// TIA Portal V15.1 export
// export: Created 2026-01-09T13:45:11.9352339Z, ExportSetting WithDefaults, WithReadOnly, DisplayName Totally Integrated Automation Portal, DisplayVersion V15.1 Update 8, DisplayName TIA Portal Openness, DisplayVersion V15.1 Update 8, DisplayName STEP 7 Professional, DisplayVersion V15.1 Update 8, DisplayName WinCC Advanced, DisplayVersion V15.1 Update 8
FUNCTION_BLOCK "1.ANALOG_INPUT"   // FB1, LAD
{ S7_Optimized_Access := 'TRUE' }
VERSION : 0.1
// stored: AutoNumber false, CodeModifiedDate 2025-09-22T19:33:21.555545Z, CompileDate 2025-09-22T19:33:35.8164831Z, CreationDate 2024-10-12T12:36:08.0193576Z, DownloadWithoutReinit false, HandleErrorsWithinBlock false, InterfaceModifiedDate 2025-09-22T19:30:11.8403437Z, IsConsistent true, IsIECCheckEnabled false, IsKnowHowProtected false, IsRetainMemResEnabled false, IsWriteProtected false, LibraryConformanceStatus The object is library-conformant., MemoryReserve 100, ModifiedDate 2025-09-22T19:33:21.555545Z, ParameterModified 2025-08-30T17:31:01.4104373Z, PLCSimAdvancedSupport false, SetENOAutomatically False, StructureModified 2025-09-22T19:30:11.8403437Z, UDAEnableTagReadback false
   VAR_INPUT
      AI : Int;
      A_MODE : Real;
      ZERO : Real;
      SPAN : Real;
      BT_ZERO : Bool;
      BT_SPAN : Bool;
      B_MANUAL : Real;
      HMI_Manual_Trigger : Bool;
   END_VAR
   VAR_OUTPUT
      W_OUT : Real;
      X_OUT : Real;
   END_VAR
   VAR RETAIN
      T_AI { ExternalAccessible := 'False'; ExternalVisible := 'False'; ExternalWritable := 'False'} : Real;
      T_AN { ExternalAccessible := 'False'; ExternalVisible := 'False'; ExternalWritable := 'False'} : Real;
      T_ZERO { ExternalAccessible := 'False'; ExternalVisible := 'False'; ExternalWritable := 'False'} : Real;
      AN_ZERO { ExternalAccessible := 'False'; ExternalVisible := 'False'; ExternalWritable := 'False'} : Real;
      T_SPAN { ExternalAccessible := 'False'; ExternalVisible := 'False'; ExternalWritable := 'False'} : Real;
      AN_SPAN { ExternalAccessible := 'False'; ExternalVisible := 'False'; ExternalWritable := 'False'} : Real;
   END_VAR
   VAR
      B_MANUAL_SAVED : Real;
      B_HAS_CHANGED : Bool;
   END_VAR
   VAR RETAIN
      IS_MANUAL_MODE : Bool;
   END_VAR
   VAR
      BT_ZERO_Raising : Bool;
      BT_SPAN_Riasing : Bool;
      MANUAL_Raissing : Bool;
      Bit_Reset_Man_Mode : Bool;
   END_VAR
   VAR_TEMP
      AI_MIN : Int;
      AI_MAX : Int;
      AN_MIN : Real;
      AN_MAX : Real;
      GT_INTEGER : DInt;
      TEMP_RESULT_DINT : DInt;
      W_OUT_MANUAL : Real;
      W_OUT_AUTO : Real;
   END_VAR
   VAR_TEMP   // added for the SCL form of the ladder/FBD networks
      _w1 : Bool;
   END_VAR
BEGIN

REGION Network 1: ANALOG MODE
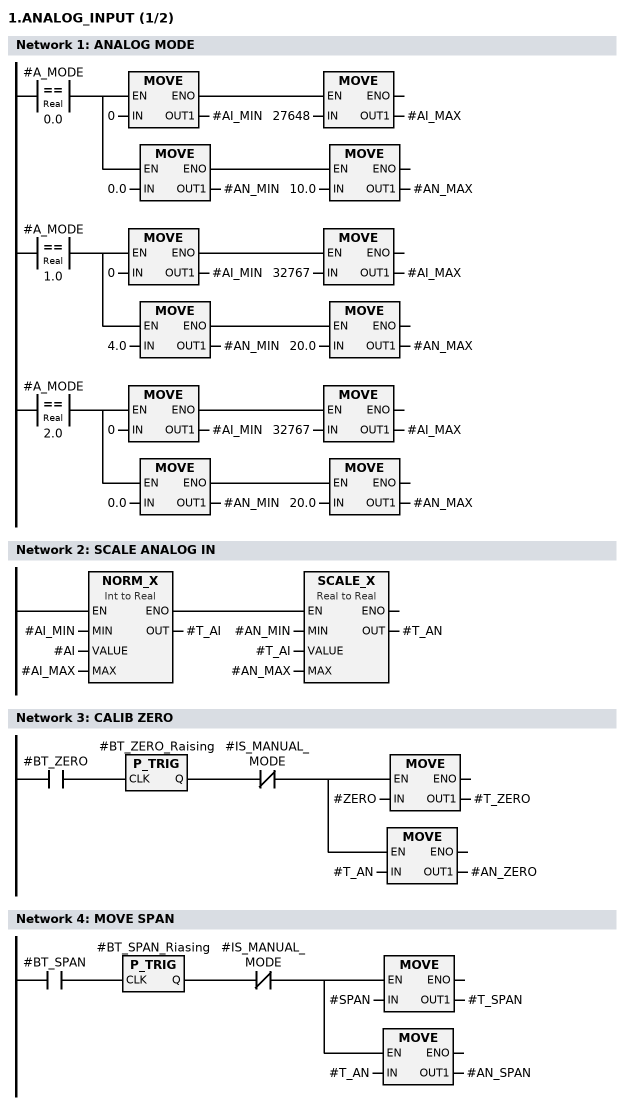
   RUNG wire#powerrail
      { S7_Templates := "SrcType := Real" } EQ_Contact(in1 := #A_MODE, in2 := 0.0)
      wire#w1
      Move(in := 0, out1 => #AI_MIN)
      Move(in := 27648, out1 => #AI_MAX)
   END_RUNG
   RUNG wire#w1
      Move(in := 0.0, out1 => #AN_MIN)
      Move(in := 10.0, out1 => #AN_MAX)
   END_RUNG
   RUNG wire#powerrail
      { S7_Templates := "SrcType := Real" } EQ_Contact(in1 := #A_MODE, in2 := 1.0)
      wire#w2
      Move(in := 0, out1 => #AI_MIN)
      Move(in := 32767, out1 => #AI_MAX)
   END_RUNG
   RUNG wire#w2
      Move(in := 4.0, out1 => #AN_MIN)
      Move(in := 20.0, out1 => #AN_MAX)
   END_RUNG
   RUNG wire#powerrail
      { S7_Templates := "SrcType := Real" } EQ_Contact(in1 := #A_MODE, in2 := 2.0)
      wire#w3
      Move(in := 0, out1 => #AI_MIN)
      Move(in := 32767, out1 => #AI_MAX)
   END_RUNG
   RUNG wire#w3
      Move(in := 0.0, out1 => #AN_MIN)
      Move(in := 20.0, out1 => #AN_MAX)
   END_RUNG
   // the same network as SCL:
   IF #A_MODE = 0.0 THEN
       #AI_MIN := 0;
       #AI_MAX := 27648;
       #AN_MIN := 0.0;
       #AN_MAX := 10.0;
   END_IF;
   IF #A_MODE = 1.0 THEN
       #AI_MIN := 0;
       #AI_MAX := 32767;
       #AN_MIN := 4.0;
       #AN_MAX := 20.0;
   END_IF;
   IF #A_MODE = 2.0 THEN
       #AI_MIN := 0;
       #AI_MAX := 32767;
       #AN_MIN := 0.0;
       #AN_MAX := 20.0;
   END_IF;
END_REGION

REGION Network 2: SCALE ANALOG IN
   RUNG wire#powerrail
      { S7_Templates := "[SrcType := Int, DestType := Real]" } Normalize(min := #AI_MIN, value := #AI, max := #AI_MAX, out => #T_AI)
      { S7_Templates := "[SrcType := Real, DestType := Real]" } Scale(min := #AN_MIN, value := #T_AI, max := #AN_MAX, out => #T_AN)
   END_RUNG
   // the same network as SCL:
   #T_AI := NORM_X(MIN := #AI_MIN, VALUE := #AI, MAX := #AI_MAX);
   #T_AN := SCALE_X(MIN := #AN_MIN, VALUE := #T_AI, MAX := #AN_MAX);
END_REGION

REGION Network 3: CALIB ZERO
   RUNG wire#powerrail
      Contact( #BT_ZERO )
      P_Trig( #BT_ZERO_Raising )
      I_Contact( #IS_MANUAL_MODE )
      wire#w1
      Move(in := #ZERO, out1 => #T_ZERO)
   END_RUNG
   RUNG wire#w1
      Move(in := #T_AN, out1 => #AN_ZERO)
   END_RUNG
   // the same network as SCL:
   #_w1 := #BT_ZERO AND NOT #BT_ZERO_Raising;   // rising edge
   #BT_ZERO_Raising := #BT_ZERO;
   IF #_w1 AND NOT #IS_MANUAL_MODE THEN
       #T_ZERO := #ZERO;
       #AN_ZERO := #T_AN;
   END_IF;
END_REGION

REGION Network 4: MOVE SPAN
   RUNG wire#powerrail
      Contact( #BT_SPAN )
      P_Trig( #BT_SPAN_Riasing )
      I_Contact( #IS_MANUAL_MODE )
      wire#w1
      Move(in := #SPAN, out1 => #T_SPAN)
   END_RUNG
   RUNG wire#w1
      Move(in := #T_AN, out1 => #AN_SPAN)
   END_RUNG
   // the same network as SCL:
   #_w1 := #BT_SPAN AND NOT #BT_SPAN_Riasing;   // rising edge
   #BT_SPAN_Riasing := #BT_SPAN;
   IF #_w1 AND NOT #IS_MANUAL_MODE THEN
       #T_SPAN := #SPAN;
       #AN_SPAN := #T_AN;
   END_IF;
END_REGION

REGION Network 5: WEIGHT OUT
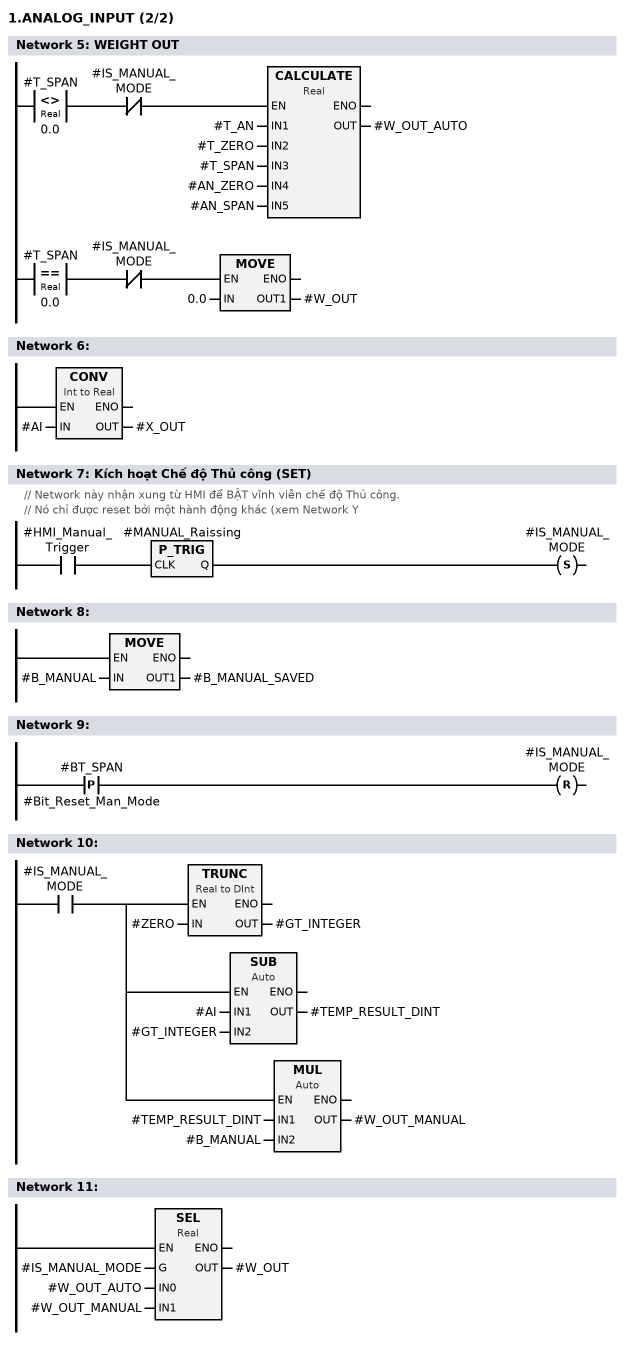
   RUNG wire#powerrail
      { S7_Templates := "SrcType := Real" } NE_Contact(in1 := #T_SPAN, in2 := 0.0)
      I_Contact( #IS_MANUAL_MODE )
      { S7_Templates := "SrcType := Real"; S7_Expression := "(IN1-IN4)/((IN5-IN4)/(IN3-IN2))" } Calculate(in1 := #T_AN, in2 := #T_ZERO, in3 := #T_SPAN, in4 := #AN_ZERO, in5 := #AN_SPAN, out => #W_OUT_AUTO)
   END_RUNG
   RUNG wire#powerrail
      { S7_Templates := "SrcType := Real" } EQ_Contact(in1 := #T_SPAN, in2 := 0.0)
      I_Contact( #IS_MANUAL_MODE )
      Move(in := 0.0, out1 => #W_OUT)
   END_RUNG
   // the same network as SCL:
   IF (#T_SPAN <> 0.0) AND NOT #IS_MANUAL_MODE THEN
       #W_OUT_AUTO := (#T_AN-#AN_ZERO)/((#AN_SPAN-#AN_ZERO)/(#T_SPAN-#T_ZERO));
   END_IF;
   IF (#T_SPAN = 0.0) AND NOT #IS_MANUAL_MODE THEN #W_OUT := 0.0; END_IF;
END_REGION

REGION Network 6
   RUNG wire#powerrail
      { S7_Templates := "[SrcType := Int, DestType := Real]" } Convert(in := #AI, out => #X_OUT)
   END_RUNG
   // the same network as SCL:
   #X_OUT := INT_TO_REAL(#AI);
END_REGION

REGION Network 7: Kích hoạt Chế độ Thủ công (SET)
   // // Network này nhận xung từ HMI để BẬT vĩnh viễn chế độ Thủ công.
   // // Nó chỉ được reset bởi một hành động khác (xem Network Y
   RUNG wire#powerrail
      Contact( #HMI_Manual_Trigger )
      P_Trig( #MANUAL_Raissing )
      S_Coil( #IS_MANUAL_MODE )
   END_RUNG
   // the same network as SCL:
   #_w1 := #HMI_Manual_Trigger AND NOT #MANUAL_Raissing;   // rising edge
   #MANUAL_Raissing := #HMI_Manual_Trigger;
   IF #_w1 THEN #IS_MANUAL_MODE := TRUE; END_IF;
END_REGION

REGION Network 8
   RUNG wire#powerrail
      Move(in := #B_MANUAL, out1 => #B_MANUAL_SAVED)
   END_RUNG
   // the same network as SCL:
   #B_MANUAL_SAVED := #B_MANUAL;
END_REGION

REGION Network 9
   RUNG wire#powerrail
      P_Contact(operand := #BT_SPAN, bit := #Bit_Reset_Man_Mode)
      R_Coil( #IS_MANUAL_MODE )
   END_RUNG
   // the same network as SCL:
   #_w1 := #BT_SPAN AND NOT #Bit_Reset_Man_Mode;   // rising edge of #BT_SPAN
   #Bit_Reset_Man_Mode := #BT_SPAN;
   IF #_w1 THEN #IS_MANUAL_MODE := FALSE; END_IF;
END_REGION

REGION Network 10
   RUNG wire#powerrail
      Contact( #IS_MANUAL_MODE )
      wire#w1
      { S7_Templates := "[SrcType := Real, DestType := DInt]" } Trunc(in := #ZERO, out => #GT_INTEGER)
   END_RUNG
   RUNG wire#w1
      Sub(in1 := #AI, in2 := #GT_INTEGER, out => #TEMP_RESULT_DINT)
   END_RUNG
   RUNG wire#w1
      Mul(in1 := #TEMP_RESULT_DINT, in2 := #B_MANUAL, out => #W_OUT_MANUAL)
   END_RUNG
   // the same network as SCL:
   IF #IS_MANUAL_MODE THEN
       #GT_INTEGER := TRUNC(#ZERO);
       #TEMP_RESULT_DINT := #AI - #GT_INTEGER;
       #W_OUT_MANUAL := #TEMP_RESULT_DINT * #B_MANUAL;
   END_IF;
END_REGION

REGION Network 11
   RUNG wire#powerrail
      { S7_Templates := "value_type := Real" } SEL(g := #IS_MANUAL_MODE, in0 := #W_OUT_AUTO, in1 := #W_OUT_MANUAL, out => #W_OUT)
   END_RUNG
   // the same network as SCL:
   #W_OUT := SEL(G := #IS_MANUAL_MODE, IN0 := #W_OUT_AUTO, IN1 := #W_OUT_MANUAL);
END_REGION
END_FUNCTION_BLOCK
